{attribute 'qualified_only'}
{attribute 'strict'}
{attribute 'to_string'}
TYPE E_DeviceStatus :
(
	Uit := 0,
	Aan := 1,
	Error:= 2
);
END_TYPE

(* stored: Version 1.1.0.1
   DUT E_DeviceStatus: Id {c4f45e34-4ad5-4662-a6fc-4f529820c7bb} *)
